TYPE E_ContactorStatus :
(
    READY := 0,         // Hazır
    OPERATING := 1,     // Çalışıyor
    INTERLOCKED := 2,   // Interlock aktif
    FAULTED := 3,       // Arızalı
    NO_CONTROL := 4,    // PLC kontrol yok
    MAINTENANCE := 5    // Bakım gerekli
);
END_TYPE

(* stored: Version 1.1.0.1, ProductVersion 3.1.4024.15
   EnumerationTextList E_ContactorStatus: Id {9c65882a-0633-4213-bc12-20182f420f68} *)
